// TIA Portal V18 export
DATA_BLOCK "_POSITIONS_RETAIN"   // DB61
{ S7_Optimized_Access := 'TRUE' }
VERSION : 0.1
// stored: AutoNumber true, DBAccessibleFromOPCUA true, IsOnlyStoredInLoadMemory false, IsRetainMemResEnabled false, IsWriteProtectedInAS false, MemoryReserve 100
   VAR RETAIN
      A1Z { S7_SetPoint := 'True'} : "typePOSMEMcalib";
      A2Y { S7_SetPoint := 'True'} : "typePOSMEMcalib";
      A3X { S7_SetPoint := 'True'} : "typePOSMEMcalib";
      A4O1 { S7_SetPoint := 'True'} : "typePOSMEMcalib";
      A5O2 { S7_SetPoint := 'True'} : "typePOSMEMcalib";
      A6Doors { S7_SetPoint := 'True'} : "typePOSMEMcalib";
   END_VAR
BEGIN
END_DATA_BLOCK
